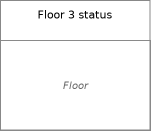
VISUALIZATION Screen3  // 151x131
    Frame (0,40 151x91)
        shows Floor(LS_Floor := MAIN.LS_Floor[3])
        OnMouseClick: change screen: Previous 
    Label (0,0 150x30), "Floor 3 status"
END_VISUALIZATION

(* stored: Version 1.1.0.1, ProductVersion 3.1.4024.11
   Visu Screen3: Id {dd9c0441-8e15-478a-8ec2-0791857908d1} *)
